PROGRAM NF_MAIN
VAR
	_context : TcoCore.TcoContextNfCompatibility;	
	_logic : NF_Logic;
END_VAR

_context.VolatileOpen();
_logic();
_context.VolatileClose();

PROPERTY Context : REFERENCE TO TcoCore.TcoContextNfCompatibility
GET
Context REF= _context;
END_GET
END_PROPERTY

END_PROGRAM

(* stored: Version 1.1.0.1, ProductVersion 3.1.4024.6
   POU NF_MAIN: Id {473a5c79-71ed-4434-b17a-54ad46fd7dad}, SpecialFunc None
   Property Context: Id {ea8b9138-b32c-43c8-a6d7-9ab2ccc07ada}
   Get Get: Id {2935880d-9d01-4fcc-9b09-0aedf712bda2} *)
